INTERFACE I_StringCollection

METHOD AddString
VAR_INPUT
	StringToAdd : T_MaxString;
END_VAR
END_METHOD

METHOD Clear : BOOL
VAR_INPUT
END_VAR
END_METHOD

PROPERTY Entries : UDINT
GET
END_GET
END_PROPERTY

END_INTERFACE

(* stored: Version 1.1.0.1, ProductVersion 3.1.4026.18
   Itf I_StringCollection: Id {948b2321-fa34-4cea-87df-e34b3cfb3399}
   Method AddString: Id {103948a8-76d9-4c96-8bd9-aed81f3079a0}
   Method Clear: Id {498f145f-cd20-4c5c-b118-f450c3eccf54}
   Property Entries: Id {e5110f88-1927-4974-88bc-b32403da1255}
   Get Get: Id {dd3a5a6a-1c74-4592-847c-c0c0c7e22eba} *)
